// TIA Portal V20 export
TYPE "LKinCtrl_typeAuxFCDiagnostics"
TITLE = typeDiagnosticsFBTemplate
   STRUCT
      status : Word;   // Status of the FB or error identification when error occurred
      subfunctionStatus : Word;   // Status or return value of called FBs, FCs and system blocks
      axisNumber : Int;   // number of the corresponding axis the error occured in or a function effecting it
      errorDetail : UDInt;   // error detail of corresponding technology object the error occured in
      stateNumber : DInt;   // State in the state machine of the FB when the error occurred
   END_STRUCT;
END_TYPE
